PROGRAM ST20_TraySequence
VAR
	arrStepStatus : ARRAY [1..100] OF STRING;
	arrStepUsedTime	: ARRAY [1..100] OF TIME;
	tonStepTimer : TON;
	iStep : INT;
	iMatching: INT;
	bStart: BOOL;
	sBarcode: STRING;
END_VAR

tonStepTimer();

bStart := (G_MachineControl.stMachineCurrentMode.AUTO_RUNNING OR
				G_MachineControl.stMachineCurrentMode.DRYRUN_RUNNING);

//New Tray Procesee
CASE iStep OF
		
	0://Ready
		IF bStart AND G_Auto.A20_bIsNewTray THEN
			G_Auto.A20_bTriggerScanner := TRUE;
			iStep := 10;
		END_IF
		
	10://Waiting scanner ack
		IF NOT G_Auto.A20_bScannerResultDone THEN
			iStep := 20;
		END_IF
		
	20://Waiting scanner result done
		IF G_Auto.A20_bScannerResultDone THEN
			sBarcode := G_Auto.A20_sScannerBarcode;
			iStep := 30;
		ELSIF G_Error.E20_BarcodeTimeout THEN
			G_Error.E20_BarcodeTimeout := FALSE;
			G_Auto.A20_bTrayReady := FALSE;
			G_Auto.A20_bMESPass := FALSE;
			G_Auto.A20_bMESCheckDone := TRUE;
			iStep := 40;
		END_IF
		
	30://Trigger check at MES
		arrStepStatus[2] := 'Step 2: Trigger Check at MES';
		G_Auto.A20_bMESPass := FALSE;
		G_Auto.A20_bMESCheckDone := FALSE;
		G_Auto.A20_bMESCheck := TRUE;
		iStep := 40;	
		
	40://Waiting check at MES done
		IF G_Auto.A20_bMESCheckDone THEN
			G_Auto.A20_bMESCheck := FALSE;
			IF G_Auto.A20_bMESPass THEN
				G_Auto.A20_bTrayReady := TRUE;
				G_Auto.A20_bIsNewTray := FALSE;
				iStep := 999;	
			ELSE
				G_Auto.A20_bTrayReady := FALSE;	
				G_Auto.A20_bTrayFinish := TRUE;
				iStep := 0;	
			END_IF
		END_IF
		
	999://Job Done
		iStep := 0;	
		
END_CASE

END_PROGRAM

(* stored: Version 1.1.0.1, ProductVersion 3.1.4024.11
   POU ST20_TraySequence: Id {540900fe-b1db-40be-acf4-286371c46f76}, SpecialFunc None *)
